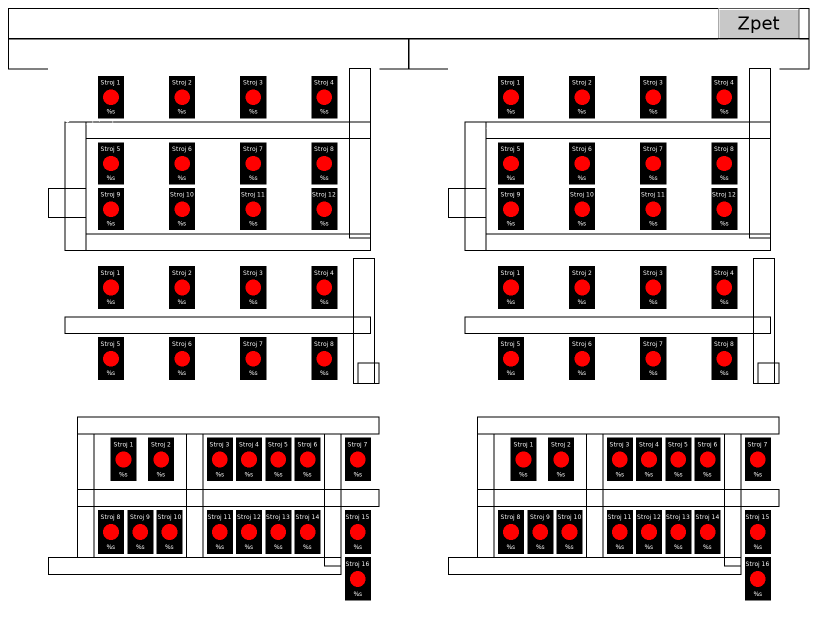
rectangle at (0,0)-(801,31): text "SLITINY"
button at (710,0)-(791,31): text "Zpet"; opens plc_vizu
rectangle at (0,30)-(401,61): text "%s"; shows PLC_PRG.Slitina[1]
rectangle at (400,30)-(801,61): text "%s"; shows PLC_PRG.Slitina[1]
embedded screen at (40,60)-(371,251): OJS_I_FS1x
embedded screen at (40,250)-(371,401): OJS_II_FS1x
embedded screen at (40,400)-(371,601): OJS_III_FS1x
embedded screen at (440,60)-(771,251): OJS_I_FS2x
embedded screen at (440,250)-(771,401): OJS_II_FS2x
embedded screen at (440,400)-(771,601): OJS_III_FS2x
*)
